// TIA Portal V20 program export: 0 tag tables, 0 data types, 1 data blocks, 3 code blocks (in call order from the OBs), 1 instance data blocks

DATA_BLOCK "InterfaceTP_C1"   // DB110
// stored: Access Published, MemoryReserve 100
   VAR
      operationOFF : Bool;   // Anlage AUS (HMI) Handbetrieb / operation ON (HMI) manual mode
      operationON : Bool;   // Anlage EIN (HMI) Automatikbetrieb / operation ON (HMI) automatic mode
      jogRight : Bool;   // Bandmotor Tippen Rechts / jog conveyor right
      jogLeft : Bool;   // Bandmotor Tippen Links / jog conveyor left
      acknowledgeFault : Bool;   // Band-Störung quittieren / acknowledge conveyor fault
      actualValue : UInt;   // Ist-Stückzahl / actual value
      setpoint : UInt := 3;   // Sollwert / setpoint value
      operation : Bool;
      conveyorFault : Bool;
   END_VAR
BEGIN
END_DATA_BLOCK

ORGANIZATION_BLOCK "Main"   // OB1, LAD, ProgramCycle
TITLE = "Main Program Sweep (Cycle)"
// stored: IsIECCheckEnabled true, SetENOAutomatically false
   VAR_INPUT
      Initial_Call : Bool;   // Initial call of this OB
      Remanence : Bool;   // =True, if remanent data are available
   END_VAR
BEGIN

REGION Network 1: New comment
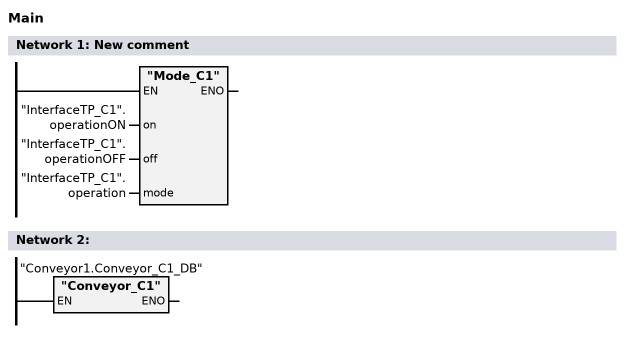
   RUNG wire#powerrail
      "Mode_C1"(on := "InterfaceTP_C1".operationON, off := "InterfaceTP_C1".operationOFF, mode := "InterfaceTP_C1".operation)
   END_RUNG
   // the same network as SCL:
   "Mode_C1"(on := "InterfaceTP_C1".operationON,
             off := "InterfaceTP_C1".operationOFF,
             mode := "InterfaceTP_C1".operation);
END_REGION

REGION Network 2
   RUNG wire#powerrail
      "Conveyor1.Conveyor_C1_DB"()
   END_RUNG
   // the same network as SCL:
   "Conveyor1.Conveyor_C1_DB"();   // "Conveyor_C1"
END_REGION
END_ORGANIZATION_BLOCK

FUNCTION "Mode_C1" : Void   // FC1, LAD
// stored: Access Published, IsIECCheckEnabled true, SetENOAutomatically false
   VAR_INPUT
      on : Bool;
      off : Bool;
   END_VAR
   VAR_IN_OUT
      mode : Bool;
   END_VAR
BEGIN

REGION Network 1
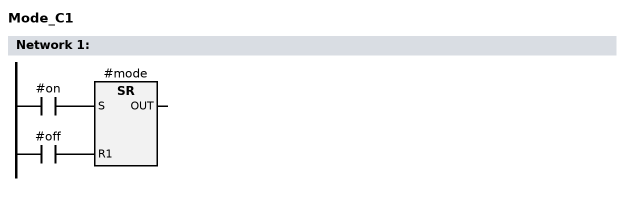
   RUNG wire#powerrail
      Contact( #on )
      S_SR(operand := #mode, r1 := wire#w1)
   END_RUNG
   RUNG wire#powerrail
      Contact( #off )
   END_RUNG wire#w1
   // the same network as SCL:
   IF #on THEN
       #mode := TRUE;   // SR flip-flop
   END_IF;
   IF #off THEN #mode := FALSE; END_IF;
END_REGION
END_FUNCTION

FUNCTION_BLOCK "Conveyor_C1"   // FB2, LAD
TITLE = New Title
// stored: Access Published, MemoryReserve 100, SetENOAutomatically false
   VAR
      jogRight : Bool;
   END_VAR
BEGIN

REGION Network 1: Run conveyor LEFT
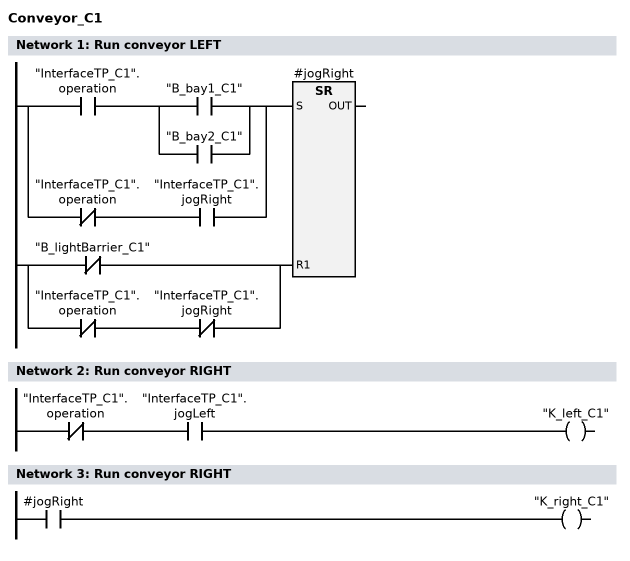
   RUNG wire#powerrail
      Contact( "InterfaceTP_C1".operation )
      wire#w1
      Contact( "B_bay1_C1" )
      wire#w2
      S_SR(operand := #jogRight, r1 := wire#w3)
   END_RUNG
   RUNG wire#w1
      Contact( "B_bay2_C1" )
   END_RUNG wire#w2
   RUNG wire#powerrail
      I_Contact( "InterfaceTP_C1".operation )
      Contact( "InterfaceTP_C1".jogRight )
   END_RUNG wire#w2
   RUNG wire#powerrail
      I_Contact( "B_lightBarrier_C1" )
   END_RUNG wire#w3
   RUNG wire#powerrail
      I_Contact( "InterfaceTP_C1".operation )
      I_Contact( "InterfaceTP_C1".jogRight )
   END_RUNG wire#w3
   // the same network as SCL:
   IF ("InterfaceTP_C1".operation AND ("B_bay1_C1" OR "B_bay2_C1")) OR (NOT "InterfaceTP_C1".operation AND "InterfaceTP_C1".jogRight) THEN
       #jogRight := TRUE;   // SR flip-flop
   END_IF;
   IF NOT "B_lightBarrier_C1" OR (NOT "InterfaceTP_C1".operation AND NOT "InterfaceTP_C1".jogRight) THEN
       #jogRight := FALSE;
   END_IF;
END_REGION

REGION Network 2: Run conveyor RIGHT
   RUNG wire#powerrail
      I_Contact( "InterfaceTP_C1".operation )
      Contact( "InterfaceTP_C1".jogLeft )
      Coil( "K_left_C1" )
   END_RUNG
   // the same network as SCL:
   "K_left_C1" := NOT "InterfaceTP_C1".operation AND "InterfaceTP_C1".jogLeft;
END_REGION

REGION Network 3: Run conveyor RIGHT
   RUNG wire#powerrail
      Contact( #jogRight )
      Coil( "K_right_C1" )
   END_RUNG
   // the same network as SCL:
   "K_right_C1" := #jogRight;
END_REGION
END_FUNCTION_BLOCK

DATA_BLOCK "Conveyor_C1_DB"   // DB3
// stored: InstanceOfName Conveyor_C1, InstanceOfType FB, Namespace Conveyor1
"Conveyor_C1"
BEGIN
END_DATA_BLOCK
